{attribute 'qualified_only'}
VAR_GLOBAL

	
	platformDir : INT := 0;

END_VAR

(* stored: Version 1.1.0.1, ProductVersion 3.1.4024.10
   GVL SensorsGVL: Id {51284672-4be5-4935-832c-7936a77761c0} *)
